// Struckig
// Copyright (C) 2022 Stefan Besler

// This program is free software: you can redistribute it and/or modify
// it under the terms of the GNU General Public License as published by
// the Free Software Foundation, either version 3 of the License, or
// (at your option) any later version.

// This program is distributed in the hope that it will be useful,
// but WITHOUT ANY WARRANTY; without even the implied warranty of
// MERCHANTABILITY or FITNESS FOR A PARTICULAR PURPOSE.  See the
// GNU General Public License for more details.
//
// You should have received a copy of the GNU General Public License
// along with THIS PROGRAM.  IF NOT, see <http://www.gnu.org/licenses/>.
/// Public interface for Struckig online trajectory generators.
/// The interface unifies access to both [Otg](xref:Struckig.Otg) (multi-DoF)
/// and [Otg1](xref:Struckig.Otg1) (single-DoF wrapper), so user code can
/// switch implementation without changing call sites.
///
/// A typical pattern is:
/// 1. Call `Cyclic` each PLC cycle.
/// 2. Monitor `State`.
/// 3. Read command setpoints from the concrete implementation outputs.
/// 4. Use `Reset` and `ValidateInput` for robust operation.
INTERFACE IOtg

/// \copydoc Struckig.Otg#AtTime
{attribute 'conditionalshow'}
METHOD AtTime
VAR_INPUT
  t : LREAL;
  new_position : POINTER TO LREAL;
  new_velocity : POINTER TO LREAL;
  new_acceleration : POINTER TO LREAL;
  new_jerk : POINTER TO LREAL;  
  new_section : POINTER TO INT;
END_VAR
END_METHOD

/// \copydoc Struckig.Otg#AtTime1
{attribute 'conditionalshow'}
METHOD AtTime1
VAR_INPUT
  t : LREAL;
  new_position : REFERENCE TO LREAL;
  new_velocity : REFERENCE TO LREAL;
  new_acceleration : REFERENCE TO LREAL;
  new_jerk : REFERENCE TO LREAL;
END_VAR
END_METHOD

/// \copydoc Struckig.Otg#Cyclic
METHOD Cyclic
VAR_INPUT
END_VAR
END_METHOD

/// \copydoc Struckig.Otg#Duration
PROPERTY Duration : LREAL
GET
END_GET
END_PROPERTY

/// \copydoc Struckig.Otg#ErrorCode
METHOD ErrorCode : TrajectoryErrorCode
VAR_INPUT
END_VAR
END_METHOD

/// \copydoc Struckig.Otg#ErrorMessage
METHOD ErrorMessage : STRING(255)
VAR_INPUT
END_VAR
END_METHOD

/// \copydoc Struckig.Otg#PassOutputToInput
METHOD PassOutputToInput
VAR_INPUT
END_VAR
END_METHOD

/// \copydoc Struckig.Otg#Reset
METHOD Reset
VAR_INPUT
END_VAR
END_METHOD

/// \copydoc Struckig.Otg#State
PROPERTY State : TrajectoryState
GET
END_GET
END_PROPERTY

/// \copydoc Struckig.Otg#ValidateInput
{attribute 'conditionalshow'}
METHOD ValidateInput : BOOL
VAR_INPUT
  checkCurrentStateWithinLimits : BOOL;
  checkTargetStateWithinLimits : BOOL;
END_VAR
END_METHOD

END_INTERFACE

(* stored: Version 1.1.0.1
   Itf IOtg: Id {a184e1a6-99b6-45c5-a545-2299a1ba3b18}
   Method AtTime: Id {41ff6a58-6de0-469e-96e7-a3465afa5f08}
   Method AtTime1: Id {0d37baef-f79a-4d1b-9576-a2376af604c9}
   Method Cyclic: Id {d26b89d9-5de1-4e69-9c66-3af979a1e1cd}
   Property Duration: Id {8c0faacd-e13f-4137-8331-68d5ef9a1818}
   Get Get: Id {279d889d-1482-438e-9f3b-c645ec4f089b}
   Method ErrorCode: Id {0747d31a-088e-4db7-8659-b8ffedb5c8af}
   Method ErrorMessage: Id {5bc8e598-ec78-4926-954b-e195d3ae2641}
   Method PassOutputToInput: Id {61e0c36c-00ec-4db9-a11d-5554a17e34af}
   Method Reset: Id {b7e13521-212e-48c5-9aa8-793af451fe62}
   Property State: Id {1fb2d035-21ef-4a96-839a-0735632d15bd}
   Get Get: Id {4517957e-24b2-4a50-b177-5b0b420d1e7f}
   Method ValidateInput: Id {a70dd70a-3498-48f3-b1ca-fd916bf70707} *)
